Universal Robots PolyScope program: test apply force.urp

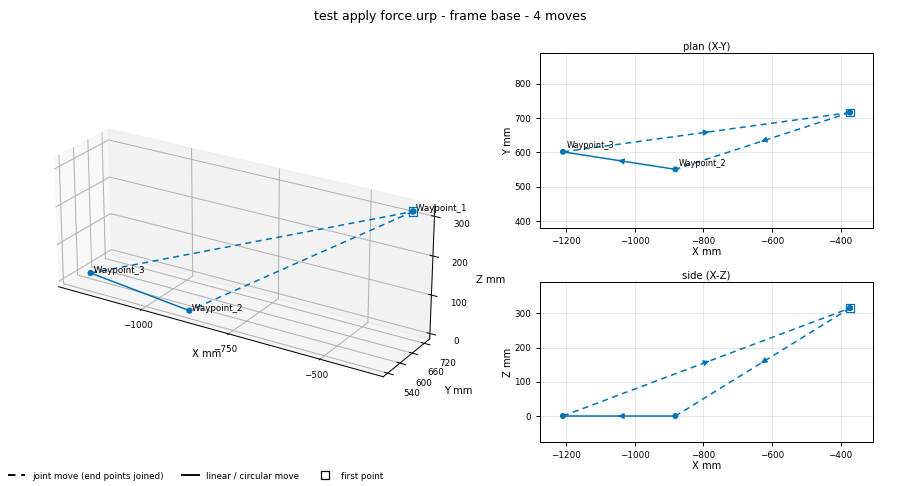
[picture p0: tool path of test apply force.urp in frame base, 4 of 4 moves have a stored position in this frame; points joined in program order, loops and branches not executed]
Program test apply force (installation=default directory=/programs createdIn=5.14.5 lastSavedIn=5.14.5 robotSerialNumber=20236801216)
Calibrated DH parameters: a=[-0.000021, -0.748897, -0.28186, -0.00004, -0.000055, 0]; d=[0.236225, -424.082933, -1564.66872, 1988.95162, 0.159094, 0.153873]; alpha=[1.570844, 0.001002, 0.000337, 1.571488, -1.569996, 0]; deltaTheta=[0, -0.516316, 5.626292, 1.173211, 0.000001, 0]
InitVariablesNode
Robot Program (runOnlyOnce=true)
  'no subprogs or variables just a force movement'
  MoveJ speed 60 deg/s, acceleration 80 deg/s^2 (useActiveTCP=true) feature=Base
    Waypoint Waypoint_1: TCP in base x=-372.868 y=716.173 z=314.672 mm, rx=1.5708 ry=0 rz=0 rad; joints [-79.16, -60.425, 105.047, -44.566, -79.226, 359.93] deg; TCP offset x=0 y=0 z=19 mm, rx=0 ry=0 rz=0 rad
    Waypoint Waypoint_2: TCP in base x=-881.132 y=550.793 z=0.591 mm, rx=1.5708 ry=0 rz=0 rad; joints [-49.438, -36.412, 90.227, -53.682, -49.494, 359.851] deg
  Wait Sleep waitTime=2
  Force Simple feature=Joint_6_name; selection=[0, 0, 1, 0, 0, 0]; wrench=[0, 0, 5, 0, 0, 0]; limitsForce=[0.15, 0.15, 0.15, 1.047198, 1.047198, 1.047198]; limitsMotion=[0.1, 0.1, 0.1, 0.349066, 0.349066, 0.349066]
    MoveP speed 20 mm/s, acceleration 1200 mm/s^2 (blendRadius=0.025 useActiveTCP=false) tcp=TCP_1_plate; feature=Base
      Waypoint Waypoint_3: TCP in base x=-1208.456 y=601.629 z=0.589 mm, rx=1.5708 ry=0 rz=0 rad; joints [-40.613, -21.006, 52.938, -31.753, -40.668, 359.801] deg
  MoveJ speed 60 deg/s, acceleration 80 deg/s^2 (useActiveTCP=true) feature=Base
    Waypoint Waypoint_1: TCP in base x=-372.868 y=716.173 z=314.672 mm, rx=1.5708 ry=0 rz=0 rad; joints [-79.16, -60.425, 105.047, -44.566, -79.226, 359.93] deg
